// LS Electric XG5000 project: P18
// PLC LSPLC

PROGRAM NewProgram (task: 스캔 프로그램)

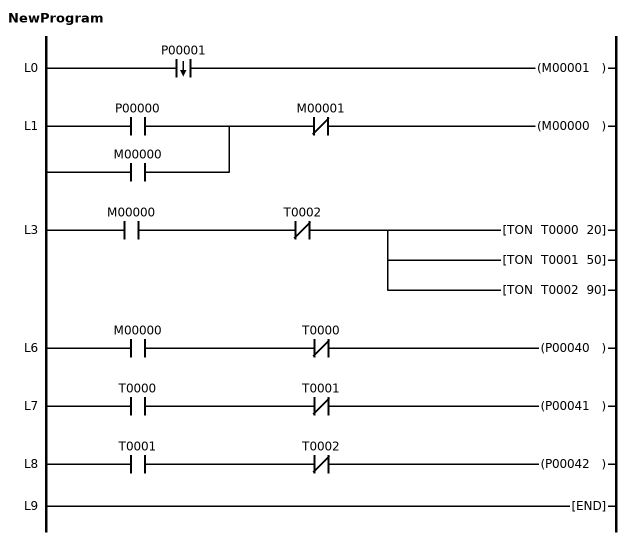
; L0
LOADN     P00001
OUT       M00001
; L1
LOAD      P00000
OR        M00000
AND NOT   M00001
OUT       M00000
; L3
LOAD      M00000
AND NOT   T0002
TON       T0000 20
TON       T0001 50
TON       T0002 90
; L6
LOAD      M00000
AND NOT   T0000
OUT       P00040
; L7
LOAD      T0000
AND NOT   T0001
OUT       P00041
; L8
LOAD      T0001
AND NOT   T0002
OUT       P00042
; L9
END